TYPE CANopenBusStatuses :
STRUCT
	///Is the device in a healthy state?
	healthStatus: HealthStatus;
END_STRUCT
END_TYPE

(* stored: Version 1.1.0.1, ProductVersion 3.1.4019.2
   DUT CANopenBusStatuses: Id {ce160452-b2b4-47e5-95d6-5959bc6185c5} *)
